// TIA Portal V18 export
// export: Created 2026-06-20T08:02:08.6526146Z, ExportSetting WithDefaults, DisplayName Totally Integrated Automation Portal, DisplayVersion V18, DisplayName TIA Portal Openness, DisplayVersion V18, DisplayName TIA Portal Version Control Interface, DisplayVersion V18, DisplayName STEP 7 Professional, DisplayVersion V18, DisplayName STEP 7 Safety, DisplayVersion V18, DisplayName WinCC Professional, DisplayVersion V18
ORGANIZATION_BLOCK "Main"   // OB1, LAD, ProgramCycle
TITLE = "Main Program Sweep (Cycle)"
{ S7_Optimized_Access := 'TRUE' }
VERSION : 0.1
// stored: AutoNumber true, IsIECCheckEnabled false, SetENOAutomatically false
   VAR_INPUT
      Initial_Call : Bool;   // Initial call of this OB
      Remanence : Bool;   // =True, if remanent data are available
   END_VAR
BEGIN

REGION Network 1: Clock 1Hz Edge Detection
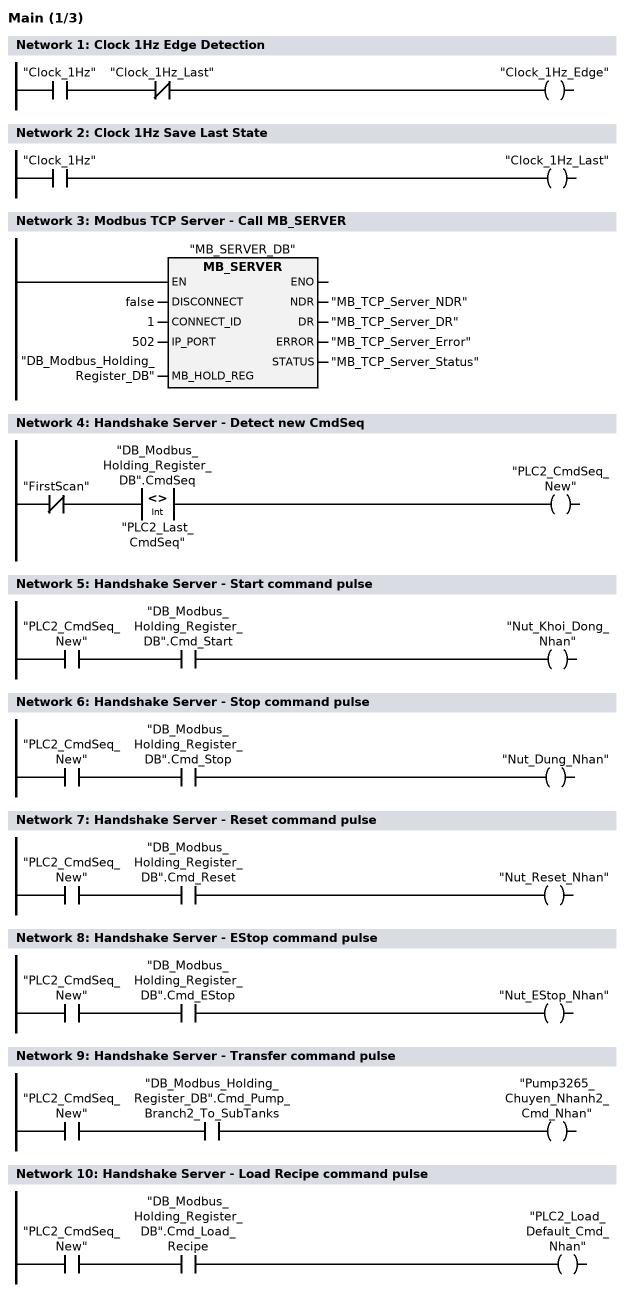
   RUNG wire#powerrail
      Contact( "Clock_1Hz" )
      I_Contact( "Clock_1Hz_Last" )
      Coil( "Clock_1Hz_Edge" )
   END_RUNG
   // the same network as SCL:
   "Clock_1Hz_Edge" := "Clock_1Hz" AND NOT "Clock_1Hz_Last";
END_REGION

REGION Network 2: Clock 1Hz Save Last State
   RUNG wire#powerrail
      Contact( "Clock_1Hz" )
      Coil( "Clock_1Hz_Last" )
   END_RUNG
   // the same network as SCL:
   "Clock_1Hz_Last" := "Clock_1Hz";
END_REGION

REGION Network 3: Modbus TCP Server - Call MB_SERVER
   RUNG wire#powerrail
      { S7_Templates := "[card1200 := 1, card1500 := 0]" } "MB_SERVER_DB".MB_SERVER(DISCONNECT := false, CONNECT_ID := 1, IP_PORT := 502, MB_HOLD_REG := "DB_Modbus_Holding_Register_DB", NDR => "MB_TCP_Server_NDR", DR => "MB_TCP_Server_DR", ERROR => "MB_TCP_Server_Error", STATUS => "MB_TCP_Server_Status")
   END_RUNG
   // the same network as SCL:
   "MB_SERVER_DB"(DISCONNECT := false,   // MB_SERVER
                  CONNECT_ID := 1,
                  IP_PORT := 502,
                  MB_HOLD_REG := "DB_Modbus_Holding_Register_DB",
                  NDR => "MB_TCP_Server_NDR",
                  DR => "MB_TCP_Server_DR",
                  ERROR => "MB_TCP_Server_Error",
                  STATUS => "MB_TCP_Server_Status");
END_REGION

REGION Network 4: Handshake Server - Detect new CmdSeq
   RUNG wire#powerrail
      I_Contact( "FirstScan" )
      { S7_Templates := "SrcType := Int" } NE_Contact(in1 := "DB_Modbus_Holding_Register_DB".CmdSeq, in2 := "PLC2_Last_CmdSeq")
      Coil( "PLC2_CmdSeq_New" )
   END_RUNG
   // the same network as SCL:
   "PLC2_CmdSeq_New" := NOT "FirstScan" AND ("DB_Modbus_Holding_Register_DB".CmdSeq <> "PLC2_Last_CmdSeq");
END_REGION

REGION Network 5: Handshake Server - Start command pulse
   RUNG wire#powerrail
      Contact( "PLC2_CmdSeq_New" )
      Contact( "DB_Modbus_Holding_Register_DB".Cmd_Start )
      Coil( "Nut_Khoi_Dong_Nhan" )
   END_RUNG
   // the same network as SCL:
   "Nut_Khoi_Dong_Nhan" := "PLC2_CmdSeq_New" AND "DB_Modbus_Holding_Register_DB".Cmd_Start;
END_REGION

REGION Network 6: Handshake Server - Stop command pulse
   RUNG wire#powerrail
      Contact( "PLC2_CmdSeq_New" )
      Contact( "DB_Modbus_Holding_Register_DB".Cmd_Stop )
      Coil( "Nut_Dung_Nhan" )
   END_RUNG
   // the same network as SCL:
   "Nut_Dung_Nhan" := "PLC2_CmdSeq_New" AND "DB_Modbus_Holding_Register_DB".Cmd_Stop;
END_REGION

REGION Network 7: Handshake Server - Reset command pulse
   RUNG wire#powerrail
      Contact( "PLC2_CmdSeq_New" )
      Contact( "DB_Modbus_Holding_Register_DB".Cmd_Reset )
      Coil( "Nut_Reset_Nhan" )
   END_RUNG
   // the same network as SCL:
   "Nut_Reset_Nhan" := "PLC2_CmdSeq_New" AND "DB_Modbus_Holding_Register_DB".Cmd_Reset;
END_REGION

REGION Network 8: Handshake Server - EStop command pulse
   RUNG wire#powerrail
      Contact( "PLC2_CmdSeq_New" )
      Contact( "DB_Modbus_Holding_Register_DB".Cmd_EStop )
      Coil( "Nut_EStop_Nhan" )
   END_RUNG
   // the same network as SCL:
   "Nut_EStop_Nhan" := "PLC2_CmdSeq_New" AND "DB_Modbus_Holding_Register_DB".Cmd_EStop;
END_REGION

REGION Network 9: Handshake Server - Transfer command pulse
   RUNG wire#powerrail
      Contact( "PLC2_CmdSeq_New" )
      Contact( "DB_Modbus_Holding_Register_DB".Cmd_Pump_Branch2_To_SubTanks )
      Coil( "Pump3265_Chuyen_Nhanh2_Cmd_Nhan" )
   END_RUNG
   // the same network as SCL:
   "Pump3265_Chuyen_Nhanh2_Cmd_Nhan" := "PLC2_CmdSeq_New" AND "DB_Modbus_Holding_Register_DB".Cmd_Pump_Branch2_To_SubTanks;
END_REGION

REGION Network 10: Handshake Server - Load Recipe command pulse
   RUNG wire#powerrail
      Contact( "PLC2_CmdSeq_New" )
      Contact( "DB_Modbus_Holding_Register_DB".Cmd_Load_Recipe )
      Coil( "PLC2_Load_Default_Cmd_Nhan" )
   END_RUNG
   // the same network as SCL:
   "PLC2_Load_Default_Cmd_Nhan" := "PLC2_CmdSeq_New" AND "DB_Modbus_Holding_Register_DB".Cmd_Load_Recipe;
END_REGION

REGION Network 11: PLC2 - Gọi logic khởi tạo recipe mặc định PLC2
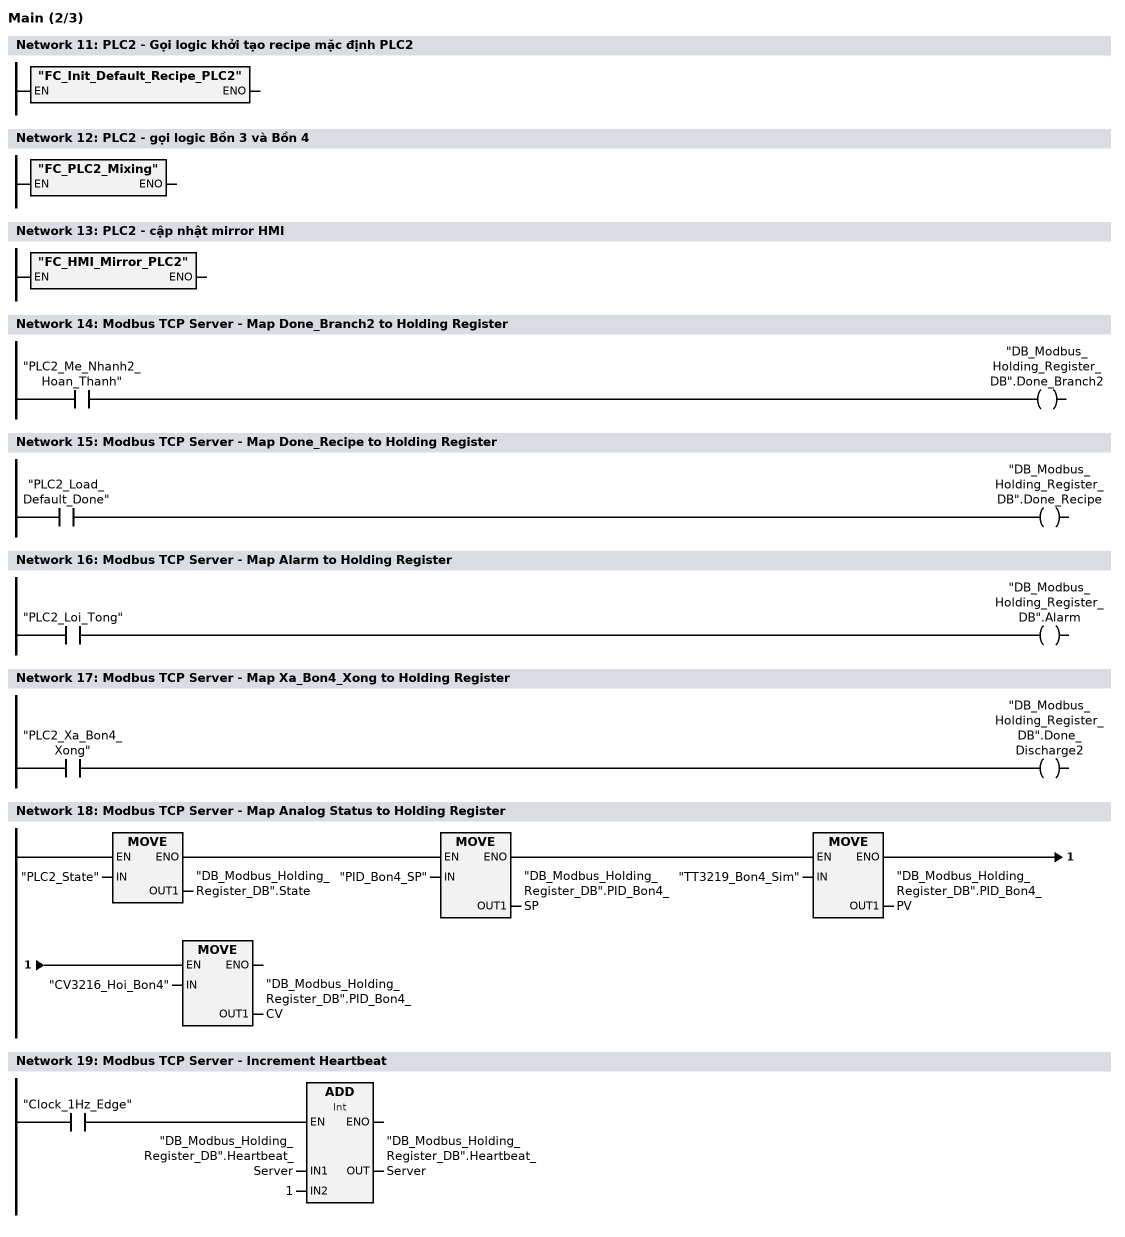
   RUNG wire#powerrail
      "FC_Init_Default_Recipe_PLC2"()
   END_RUNG
   // the same network as SCL:
   "FC_Init_Default_Recipe_PLC2"();
END_REGION

REGION Network 12: PLC2 - gọi logic Bồn 3 và Bồn 4
   RUNG wire#powerrail
      "FC_PLC2_Mixing"()
   END_RUNG
   // the same network as SCL:
   "FC_PLC2_Mixing"();
END_REGION

REGION Network 13: PLC2 - cập nhật mirror HMI
   RUNG wire#powerrail
      "FC_HMI_Mirror_PLC2"()
   END_RUNG
   // the same network as SCL:
   "FC_HMI_Mirror_PLC2"();
END_REGION

REGION Network 14: Modbus TCP Server - Map Done_Branch2 to Holding Register
   RUNG wire#powerrail
      Contact( "PLC2_Me_Nhanh2_Hoan_Thanh" )
      Coil( "DB_Modbus_Holding_Register_DB".Done_Branch2 )
   END_RUNG
   // the same network as SCL:
   "DB_Modbus_Holding_Register_DB".Done_Branch2 := "PLC2_Me_Nhanh2_Hoan_Thanh";
END_REGION

REGION Network 15: Modbus TCP Server - Map Done_Recipe to Holding Register
   RUNG wire#powerrail
      Contact( "PLC2_Load_Default_Done" )
      Coil( "DB_Modbus_Holding_Register_DB".Done_Recipe )
   END_RUNG
   // the same network as SCL:
   "DB_Modbus_Holding_Register_DB".Done_Recipe := "PLC2_Load_Default_Done";
END_REGION

REGION Network 16: Modbus TCP Server - Map Alarm to Holding Register
   RUNG wire#powerrail
      Contact( "PLC2_Loi_Tong" )
      Coil( "DB_Modbus_Holding_Register_DB".Alarm )
   END_RUNG
   // the same network as SCL:
   "DB_Modbus_Holding_Register_DB".Alarm := "PLC2_Loi_Tong";
END_REGION

REGION Network 17: Modbus TCP Server - Map Xa_Bon4_Xong to Holding Register
   RUNG wire#powerrail
      Contact( "PLC2_Xa_Bon4_Xong" )
      Coil( "DB_Modbus_Holding_Register_DB".Done_Discharge2 )
   END_RUNG
   // the same network as SCL:
   "DB_Modbus_Holding_Register_DB".Done_Discharge2 := "PLC2_Xa_Bon4_Xong";
END_REGION

REGION Network 18: Modbus TCP Server - Map Analog Status to Holding Register
   RUNG wire#powerrail
      { S7_GenerateENO := "TRUE" } Move(in := "PLC2_State", out1 => "DB_Modbus_Holding_Register_DB".State)
      { S7_GenerateENO := "TRUE" } Move(in := "PID_Bon4_SP", out1 => "DB_Modbus_Holding_Register_DB".PID_Bon4_SP)
      { S7_GenerateENO := "TRUE" } Move(in := "TT3219_Bon4_Sim", out1 => "DB_Modbus_Holding_Register_DB".PID_Bon4_PV)
      { S7_GenerateENO := "TRUE" } Move(in := "CV3216_Hoi_Bon4", out1 => "DB_Modbus_Holding_Register_DB".PID_Bon4_CV)
   END_RUNG
   // the same network as SCL:
   // ENO of a box is taken as its EN; it also drops when the box reports an error
   "DB_Modbus_Holding_Register_DB".State := "PLC2_State";
   "DB_Modbus_Holding_Register_DB".PID_Bon4_SP := "PID_Bon4_SP";
   "DB_Modbus_Holding_Register_DB".PID_Bon4_PV := "TT3219_Bon4_Sim";
   "DB_Modbus_Holding_Register_DB".PID_Bon4_CV := "CV3216_Hoi_Bon4";
END_REGION

REGION Network 19: Modbus TCP Server - Increment Heartbeat
   RUNG wire#powerrail
      Contact( "Clock_1Hz_Edge" )
      { S7_Templates := "SrcType := Int"; S7_GenerateENO := "TRUE" } Add(in1 := "DB_Modbus_Holding_Register_DB".Heartbeat_Server, in2 := 1, out => "DB_Modbus_Holding_Register_DB".Heartbeat_Server)
   END_RUNG
   // the same network as SCL:
   IF "Clock_1Hz_Edge" THEN
       "DB_Modbus_Holding_Register_DB".Heartbeat_Server := "DB_Modbus_Holding_Register_DB".Heartbeat_Server + 1;
   END_IF;
END_REGION

REGION Network 20: Modbus TCP Server - Monitor Heartbeat Change
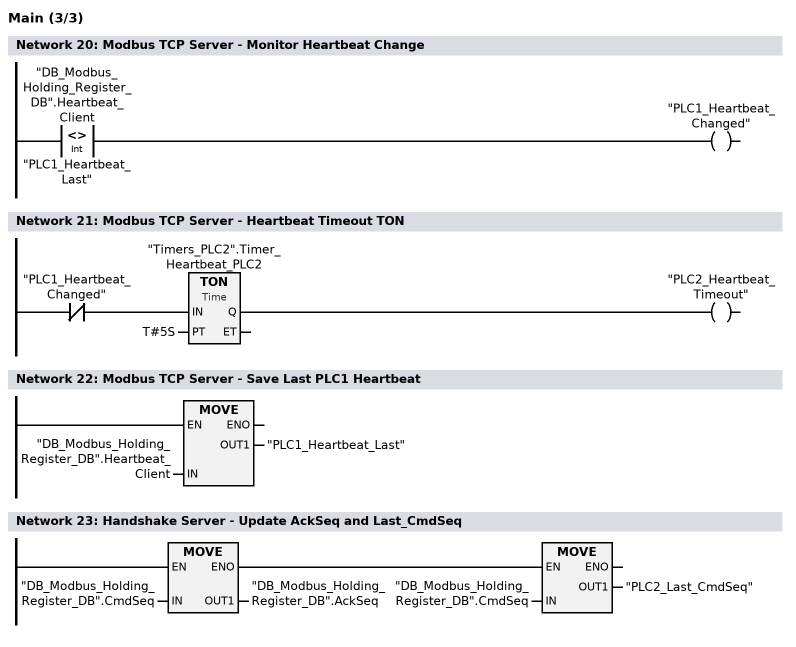
   RUNG wire#powerrail
      { S7_Templates := "SrcType := Int" } NE_Contact(in1 := "DB_Modbus_Holding_Register_DB".Heartbeat_Client, in2 := "PLC1_Heartbeat_Last")
      Coil( "PLC1_Heartbeat_Changed" )
   END_RUNG
   // the same network as SCL:
   "PLC1_Heartbeat_Changed" := "DB_Modbus_Holding_Register_DB".Heartbeat_Client <> "PLC1_Heartbeat_Last";
END_REGION

REGION Network 21: Modbus TCP Server - Heartbeat Timeout TON
   RUNG wire#powerrail
      I_Contact( "PLC1_Heartbeat_Changed" )
      { S7_Templates := "time_type := Time" } "Timers_PLC2".Timer_Heartbeat_PLC2.TON(pt := T#5S, et =>)
      Coil( "PLC2_Heartbeat_Timeout" )
   END_RUNG
   // the same network as SCL:
   "Timers_PLC2".Timer_Heartbeat_PLC2.TON(IN := NOT "PLC1_Heartbeat_Changed", PT := T#5S);
   "PLC2_Heartbeat_Timeout" := "Timers_PLC2".Timer_Heartbeat_PLC2.Q;
END_REGION

REGION Network 22: Modbus TCP Server - Save Last PLC1 Heartbeat
   RUNG wire#powerrail
      { S7_GenerateENO := "TRUE" } Move(in := "DB_Modbus_Holding_Register_DB".Heartbeat_Client, out1 => "PLC1_Heartbeat_Last")
   END_RUNG
   // the same network as SCL:
   "PLC1_Heartbeat_Last" := "DB_Modbus_Holding_Register_DB".Heartbeat_Client;
END_REGION

REGION Network 23: Handshake Server - Update AckSeq and Last_CmdSeq
   RUNG wire#powerrail
      { S7_GenerateENO := "TRUE" } Move(in := "DB_Modbus_Holding_Register_DB".CmdSeq, out1 => "DB_Modbus_Holding_Register_DB".AckSeq)
      { S7_GenerateENO := "TRUE" } Move(in := "DB_Modbus_Holding_Register_DB".CmdSeq, out1 => "PLC2_Last_CmdSeq")
   END_RUNG
   // the same network as SCL:
   // ENO of a box is taken as its EN; it also drops when the box reports an error
   "DB_Modbus_Holding_Register_DB".AckSeq := "DB_Modbus_Holding_Register_DB".CmdSeq;
   "PLC2_Last_CmdSeq" := "DB_Modbus_Holding_Register_DB".CmdSeq;
END_REGION
END_ORGANIZATION_BLOCK
